% RSLogix 500 project Project_3.RSS, saved by version 8.30.00.16 %
PROJECT "UNTITLED"    % processor: Bul.1763 MicroLogix 1100 Series B %

PROGRAM FILES
  LAD 2 "BARCODE"  5 rungs
  LAD 3 "DECISION"  4 rungs
  LAD 4 "STRG CLU"  2 rungs

DATA FILES
  O0 OUTPUT  4 elements
  I1 INPUT  6 elements
  S2 STATUS  66 elements
  B3 BINARY  1 elements
  T4 TIMER  1 elements
  C5 COUNTER  1 elements
  R6 CONTROL  1 elements
  N7 INTEGER  7 elements
  F8 FLOAT  1 elements
  ST9 STRING  4 elements

LADDER 2 "BARCODE"
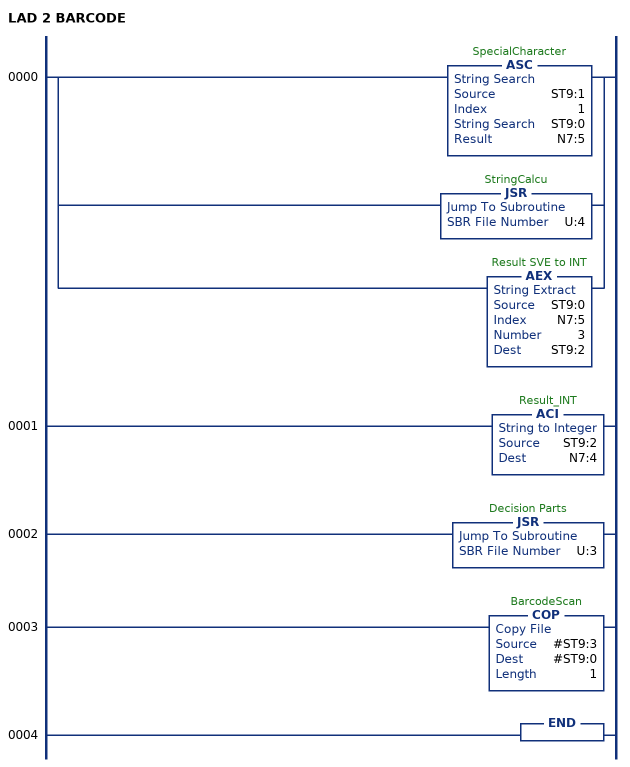
% Rung: 0 %
SOR BST ASC ST9:1 1 ST9:0 N7:5 NXB JSR U:4 NXB AEX ST9:0 N7:5 3 ST9:2 BND EOR
%   ST9:1  "SpecialCharacter" %
%   ST9:0  "BarcodeScan" %
%   N7:5  "ResultString" %
%   U:4  "StringCalcu" %
%   ST9:2  "Result SVE to INT" %
% Rung: 1 %
SOR ACI ST9:2 N7:4 EOR
%   ST9:2  "Result SVE to INT" %
%   N7:4  "Result_INT" %
% Rung: 2 %
SOR JSR U:3 EOR
%   U:3  "Decision Parts" %
% Rung: 3 %
SOR COP #ST9:3 #ST9:0 1 EOR
%   ST9:3  "Reset" %
%   ST9:0  "BarcodeScan" %
% Rung: 4 %
SOR END EOR

LADDER 3 "DECISION"
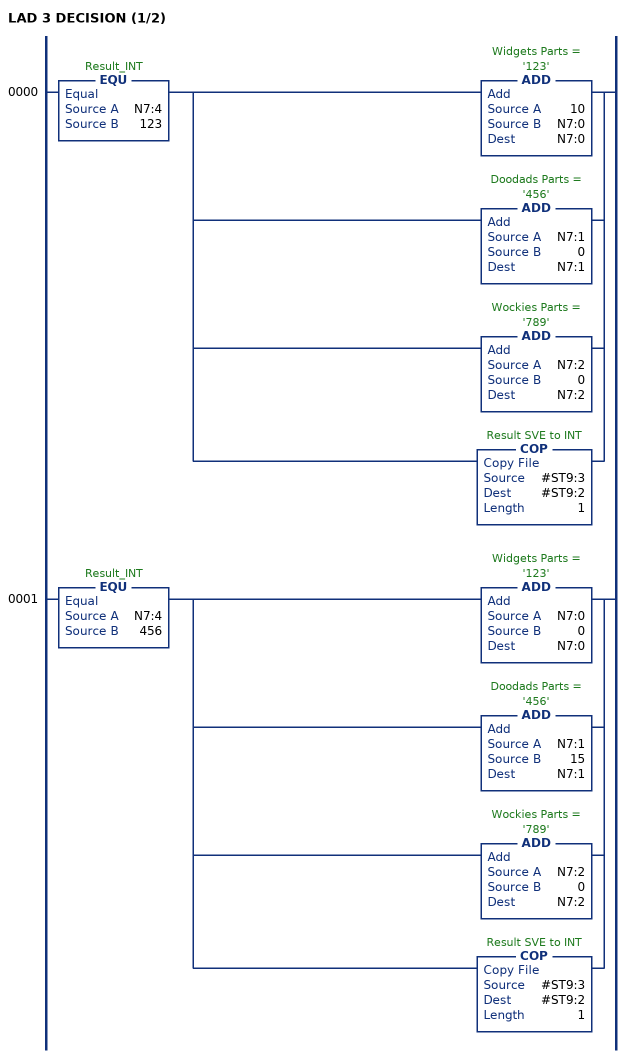
% Rung: 0 %
SOR EQU N7:4 123 BST ADD 10 N7:0 N7:0 NXB ADD N7:1 0 N7:1 NXB ADD N7:2 0 N7:2 NXB COP #ST9:3 #ST9:2 1 BND EOR
%   N7:4  "Result_INT" %
%   N7:0  "Widgets Parts = '123'" %
%   N7:1  "Doodads Parts = '456'" %
%   N7:2  "Wockies Parts = '789'" %
%   ST9:3  "Reset" %
%   ST9:2  "Result SVE to INT" %
% Rung: 1 %
SOR EQU N7:4 456 BST ADD N7:0 0 N7:0 NXB ADD N7:1 15 N7:1 NXB ADD N7:2 0 N7:2 NXB COP #ST9:3 #ST9:2 1 BND EOR
%   N7:4  "Result_INT" %
%   N7:0  "Widgets Parts = '123'" %
%   N7:1  "Doodads Parts = '456'" %
%   N7:2  "Wockies Parts = '789'" %
%   ST9:3  "Reset" %
%   ST9:2  "Result SVE to INT" %

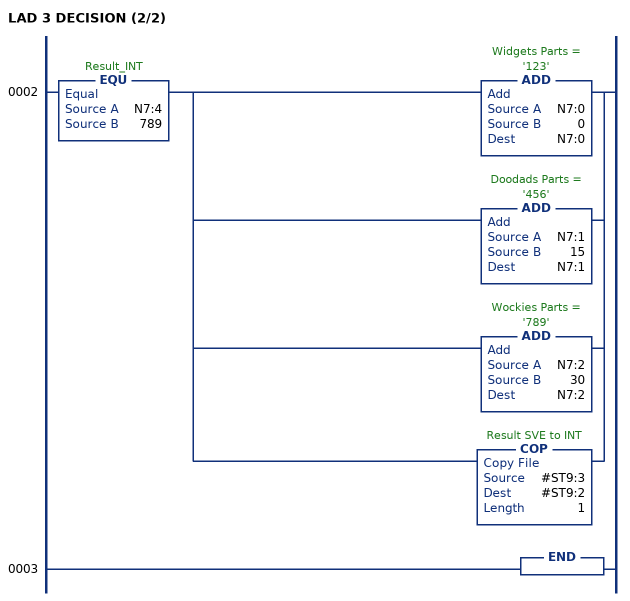
% Rung: 2 %
SOR EQU N7:4 789 BST ADD N7:0 0 N7:0 NXB ADD N7:1 15 N7:1 NXB ADD N7:2 30 N7:2 NXB COP #ST9:3 #ST9:2 1 BND EOR
%   N7:4  "Result_INT" %
%   N7:0  "Widgets Parts = '123'" %
%   N7:1  "Doodads Parts = '456'" %
%   N7:2  "Wockies Parts = '789'" %
%   ST9:3  "Reset" %
%   ST9:2  "Result SVE to INT" %
% Rung: 3 %
SOR END EOR

LADDER 4 "STRG CLU"
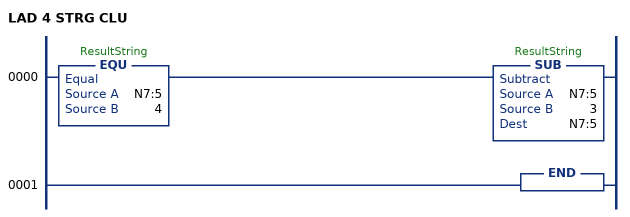
% Rung: 0 %
SOR EQU N7:5 4 SUB N7:5 3 N7:5 EOR
%   N7:5  "ResultString" %
% Rung: 1 %
SOR END EOR

OTHER DOCUMENTED ADDRESSES
  B3:0/0  "Return"
  B3:0/3  "Start"
  B3:0/4  "Switch"
  B3:0/5  "ONS"
  B3:0/6  "Switch"
  N7:6  "test"
  U:2  "ResultString"

DATA TABLE (non-zero values as saved)
DATA ST9
% ST9:0 % "123-10:1"
% ST9:1 % "-"
